// TIA Portal V20 export
TYPE "LBP_typeHandwheel"
TITLE = Handwheel image / Image de la manivelle
// User data type for handwheel / Type de données utilisateur pour manivelle
   STRUCT
      handWheel1 : Int;
      handWheel2 : Int;
   END_STRUCT;
END_TYPE
